# EPICS autosave request: iocBoot/iocImg/cam_auto_settings.req
file "aravisGigE_settings.req",     P=$(P),  R=det1:
file "NDStdArrays_settings.req",    P=$(P),  R=image1:
file "commonPlugin_settings.req",   P=$(P)
